//{attribute 'qualified_only'}
//{attribute 'strict'}
{attribute 'to_string'}
TYPE Thankfillingenum :
(
	IDLlE := 0,
	FILLING  := 1,
	FULL  := 2,
	DRAINING  := 3,
	FAULT  := 4
);
END_TYPE

(* stored: Version 1.1.0.1
   DUT Thankfillingenum: Id {9f624e8b-3c0b-4056-a319-d53692b4f024} *)
